FUNCTION_BLOCK FB_ConveyorMotor
VAR
	bStart			AT%Q*		:BOOL;	//Output to turn motor on
	bFuse			AT%I*		:BOOL;	//Motor is Running
	bThermistor		AT%I*		:BOOL;	//Motor is Ok
END_VAR

PROPERTY Fuse : BOOL
GET
Fuse:=bFuse;
END_GET
END_PROPERTY

METHOD RunMotor : BOOL
VAR
	Motor	:FB_ConveyorMotor;
END_VAR
IF Motor.bStart AND NOT FUSE AND NOT Thermistor THEN
	RunMotor:=TRUE;
	ELSE
	RunMotor:=FALSE;
END_IF
END_METHOD

PROPERTY Start : BOOL
SET
bStart:=Start;
END_SET
END_PROPERTY

PROPERTY Thermistor : BOOL
GET
Thermistor:=bThermistor;
END_GET
END_PROPERTY

END_FUNCTION_BLOCK

(* stored: Version 1.1.0.1, ProductVersion 3.1.4024.12
   POU FB_ConveyorMotor: Id {fc0b36fa-73c9-45f9-8d9a-ec2e7801497a}, SpecialFunc None
   Property Fuse: Id {2d6fa50e-bf84-4d88-9639-7953081bf742}
   Get Get: Id {4c4141f4-d864-4f70-9931-a1d7b4fe74eb}
   Method RunMotor: Id {93d74e23-87ee-4e6a-bcc2-7dbead150d0e}
   Property Start: Id {8dd4e5fe-37f4-41c8-9bf2-6aaf2b742374}
   Set Set: Id {b270632a-1bdd-475b-86fb-96186f35a726}
   Property Thermistor: Id {38752e4c-53e8-4720-be90-1dc76faae53d}
   Get Get: Id {95c6ac38-0f77-4bc6-ab86-a79efd819dde} *)
